// TIA Portal V19 export
TYPE "LEXCHANGETRAY_typeConstraintRollerEm_xPositionAxis_controlNode"
// stored: Access Published
   STRUCT
      axisControlControlNode : "LBC_typeAxisSimpleControlNode_1";
      xPosmonitor { S7_SetPoint := 'True'} : "LEXCHANGETRAY_typeConstraintRollerEm_xPositionAxis_monitor";
      posPoint { S7_SetPoint := 'True'} : Array[0..99] of "typePosAxisParameter";
      posIndex : Int;
   END_STRUCT;
END_TYPE
